(* IEC 61131-3 sources: BrdkAlarm/, 3 files *)

(* ---- Types.typ ---- *)
TYPE
	BrdkAlarmControlInternalType : 	STRUCT
		MpComConfigBasic_0 : MpComConfigBasic; (*Function block for reading and writing alarm configuration*)
		instanceID : UDINT; (*Unique ID of the alarm when active*)
		TON_delay : TON; (*AlarmDelay timer*)
		alarmActive : BOOL; (*Internal state of the alarm when taking delay and inhibit into account*)
		alarmCfgName : STRING[255]; (*Internal name of the alarm config*)
		alarmInstanceName : STRING[255]; (*Internal name of the alarm instance*)
		acknowledgeOld : BOOL; (*Edge detection*)
		confirmOld : BOOL; (*Edge detection*)
		errorResetOld : BOOL; (*Edge detection*)
	END_STRUCT;
END_TYPE

(* ---- BrdkAlarm.fun ---- *)
FUNCTION_BLOCK BrdkAlarmControl (*Function block for optionally adding an alarm configuration and controlling the alarm*) (*$GROUP=User,$CAT=User,$GROUPICON=User.png,$CATICON=User.png*)
	VAR_INPUT
		Enable : BOOL; (*Enable the function block*)
		MpLinkCore : REFERENCE TO MpComIdentType; (*MpLink of the MpAlarmX Core configuration *)
		MpLinkList : REFERENCE TO MpComIdentType; (*MpLink of the MpAlarmX List configuration *)
		AlarmConfig : MpAlarmXCfgListAlarmType := (Code:=0,Severity:=1,Behavior:=(Type:=mpALARMX_CFG_LIST_PERSISTENT,Edge:=(Confirm:=mpALARMX_CFG_LIST_CFM_DISABLED,MultipleInstances:=TRUE,ReactionWhilePending:=TRUE,Retain:=FALSE,Asynchronous:=FALSE,DataUpdate:=(Activation:=(Timestamp:=FALSE,Snippets:=FALSE)),HistoryReport:=(InactiveToActive:=TRUE,UnacknowledgedToAcknowledged:=TRUE,AcknowledgedToUnacknowledged:=FALSE,UnconfirmedToConfirmed:=TRUE,ConfirmedToUnconfirmed:=FALSE)),Persistent:=(Acknowledge:=mpALARMX_CFG_LIST_ACK_REQ,Confirm:=mpALARMX_CFG_LIST_CFM_DISABLED,MultipleInstances:=FALSE,ReactionWhilePending:=TRUE,Retain:=FALSE,Asynchronous:=FALSE,DataUpdate:=(Activation:=(Timestamp:=FALSE,Snippets:=FALSE)),HistoryReport:=(InactiveToActive:=TRUE,ActiveToInactive:=FALSE,UnacknowledgedToAcknowledged:=TRUE,AcknowledgedToUnacknowledged:=FALSE,UnconfirmedToConfirmed:=TRUE,ConfirmedToUnconfirmed:=FALSE,Update:=FALSE)),UserDefined:=(AutoReset:=FALSE,Acknowledge:=mpALARMX_CFG_LIST_ACK_REQ,Confirm:=mpALARMX_CFG_LIST_CFM_DISABLED,MultipleInstances:=FALSE,ReactionWhilePending:=TRUE,Retain:=FALSE,Asynchronous:=FALSE,DataUpdate:=(Activation:=(Timestamp:=FALSE,Snippets:=FALSE)),HistoryReport:=(InactiveToActive:=TRUE,ActiveToInactive:=TRUE,UnacknowledgedToAcknowledged:=TRUE,AcknowledgedToUnacknowledged:=FALSE,UnconfirmedToConfirmed:=TRUE,ConfirmedToUnconfirmed:=FALSE,Update:=FALSE)),Level:=(Acknowledge:=mpALARMX_CFG_LIST_ACK_REQ,Confirm:=mpALARMX_CFG_LIST_CFM_DISABLED,ReactionWhilePending:=TRUE,HistoryReport:=(InactiveToActive:=TRUE,ActiveToInactive:=FALSE,UnacknowledgedToAcknowledged:=TRUE,AcknowledgedToUnacknowledged:=FALSE,UnconfirmedToConfirmed:=TRUE,ConfirmedToUnconfirmed:=FALSE,Update:=FALSE),Monitoring:=(Exclusive:=TRUE,LowLimit:=(Type:=mpALARMX_CFG_LIST_LIMIT_DISABLED,LimitStatic:=(Limit:=0)),LowLowLimit:=(Type:=mpALARMX_CFG_LIST_LIMIT_DISABLED,LimitStatic:=(Limit:=0)),HighLimit:=(Type:=mpALARMX_CFG_LIST_LIMIT_DISABLED,LimitStatic:=(Limit:=0)),HighHighLimit:=(Type:=mpALARMX_CFG_LIST_LIMIT_DISABLED,LimitStatic:=(Limit:=0)),Settings:=(Type:=mpALARMX_CFG_LIST_STATIC,Static:=(Delay:=0,Hysteresis:=0)))),Deviation:=(Acknowledge:=mpALARMX_CFG_LIST_ACK_REQ,Confirm:=mpALARMX_CFG_LIST_CFM_DISABLED,ReactionWhilePending:=TRUE,HistoryReport:=(InactiveToActive:=TRUE,ActiveToInactive:=FALSE,UnacknowledgedToAcknowledged:=TRUE,AcknowledgedToUnacknowledged:=FALSE,UnconfirmedToConfirmed:=TRUE,ConfirmedToUnconfirmed:=FALSE,Update:=FALSE),Monitoring:=(Exclusive:=TRUE,LowLimit:=(Type:=mpALARMX_CFG_LIST_LIMIT_DISABLED,LimitStatic:=(Limit:=0)),LowLowLimit:=(Type:=mpALARMX_CFG_LIST_LIMIT_DISABLED,LimitStatic:=(Limit:=0)),HighLimit:=(Type:=mpALARMX_CFG_LIST_LIMIT_DISABLED,LimitStatic:=(Limit:=0)),HighHighLimit:=(Type:=mpALARMX_CFG_LIST_LIMIT_DISABLED,LimitStatic:=(Limit:=0)),Settings:=(Type:=mpALARMX_CFG_LIST_STATIC,Static:=(Delay:=0,Hysteresis:=0)))),RateOfChange:=(Acknowledge:=mpALARMX_CFG_LIST_ACK_REQ,Confirm:=mpALARMX_CFG_LIST_CFM_DISABLED,ReactionWhilePending:=TRUE,HistoryReport:=(InactiveToActive:=TRUE,ActiveToInactive:=FALSE,UnacknowledgedToAcknowledged:=TRUE,AcknowledgedToUnacknowledged:=FALSE,UnconfirmedToConfirmed:=TRUE,ConfirmedToUnconfirmed:=FALSE,Update:=FALSE),Monitoring:=(Exclusive:=TRUE,LowLimit:=(Type:=mpALARMX_CFG_LIST_LIMIT_DISABLED,LimitStatic:=(Limit:=0)),LowLowLimit:=(Type:=mpALARMX_CFG_LIST_LIMIT_DISABLED,LimitStatic:=(Limit:=0)),HighLimit:=(Type:=mpALARMX_CFG_LIST_LIMIT_DISABLED,LimitStatic:=(Limit:=0)),HighHighLimit:=(Type:=mpALARMX_CFG_LIST_LIMIT_DISABLED,LimitStatic:=(Limit:=0)),Settings:=(Type:=mpALARMX_CFG_LIST_TIM_STATIC,Static:=(Delay:=0,TimeConstant:=0)))),Discrete:=(Acknowledge:=mpALARMX_CFG_LIST_ACK_REQ,Confirm:=mpALARMX_CFG_LIST_CFM_DISABLED,ReactionWhilePending:=TRUE,HistoryReport:=(InactiveToActive:=TRUE,ActiveToInactive:=FALSE,UnacknowledgedToAcknowledged:=TRUE,AcknowledgedToUnacknowledged:=FALSE,UnconfirmedToConfirmed:=TRUE,ConfirmedToUnconfirmed:=FALSE,Update:=FALSE),Monitoring:=(Trigger:=(NumberOfAlarmValues:=0)))),Disable:=FALSE); (*Configuration of a new alarm to the list*)
		Name : STRING[255]; (*Name of an existing alarm instance. Use AlarmConfig.Name input to configure a new alarm at runtime. Leave Name empty to use AlarmConfig.Name as instance name.*)
		NameInConfig : STRING[255]; (*Name of an existing alarm configuration if different than alarm instance name (input: Name). If left empty Name will be used. NameInConfig is necessary if tokens like {1} are used.*)
		Condition : BOOL; (*State of the alarm condition. If TRUE the alarm will be set after the delay if not inhibitted. If FALSE the alarm will be reset*)
		Delay : TIME; (*Alarm Delay. The alarm will be triggered after the delay if Condition is TRUE and Inhibit is FALSE*)
		Inhibit : BOOL; (*Inhibits the alarm from being set. If already active it will be reset*)
		Acknowledge : BOOL; (*Acknowledge the alarm*)
		Confirm : BOOL; (*Confirm the alarm*)
		ErrorReset : BOOL; (*Resets error(s) on the MpComConfigBasic if it fails to read or save alarm config*)
	END_VAR
	VAR_OUTPUT
		Active : BOOL; (*Active when the function block is enabled*)
		AlarmActive : BOOL; (*TRUE if alarm has been set and FALSE if alarm has been reset*)
		InstanceID : UDINT; (*InstanceID of the alarm if Active*)
		StatusID : DINT; (*ID of the status from MpComConfigBasic*)
		Info : MpAlarmXCfgListAlarmType; (*Alarm config info*)
		Error : BOOL; (*An error is active and must be reset*)
	END_VAR
	VAR
		internal : BrdkAlarmControlInternalType; (*Internal type*)
		state : UINT; (*Internal state of the function block*)
	END_VAR
END_FUNCTION_BLOCK

(* ---- Constants.var ---- *)
VAR CONSTANT

END_VAR
